INTERFACE I_EventReaction EXTENDS I_Resettable

METHOD GetHighestActiveEventReaction : DINT;
END_METHOD

METHOD SetEventReactions
VAR_INPUT
	Verbose	 : DINT := 0;
	Info	 : DINT := 1;
	Warning	 : DINT := 2;
	Error	 : DINT := 3;
	Critical : DINT := 4;
END_VAR
END_METHOD

END_INTERFACE

(* stored: Version 1.1.0.1, ProductVersion 3.1.4026.18
   Itf I_EventReaction: Id {2d3762dd-5d80-4ddd-8558-4e0b9ee44a56}
   Method GetHighestActiveEventReaction: Id {26c945db-abca-484f-a18c-e9a17a338df6}
   Method SetEventReactions: Id {91c44206-9ee8-4d78-984e-96e2b8b818b9} *)
